# EPICS autosave request: mrfApp/Db/evg-vme.inc.req
$(P)$(R)IRQ:DataBuffer:Enabled.VAL
$(P)$(R)IRQ:Enabled.VAL
$(P)$(R)IRQ:EventFIFOFull:Enabled.VAL
$(P)$(R)IRQ:External:Enabled.VAL
$(P)$(R)IRQ:RXViolation:Enabled.VAL
$(P)$(R)IRQ:SeqRAM0Start:Enabled.VAL
$(P)$(R)IRQ:SeqRAM1Start:Enabled.VAL
$(P)$(R)IRQ:SeqRAM0Stop:Enabled.VAL
$(P)$(R)IRQ:SeqRAM1Stop:Enabled.VAL
